Staubli VAL3: start.pgx

program start()
begin
  call create(0,"detect")
end
